{attribute 'GeneratedUsingTerminal: AT2041-0250-0020'}
{attribute addProperty BoxType "AT2041-0250-0020"}
{attribute addProperty Id "A_0102_AT2041_5250_0019_AT2041_5250AT2041_01D6DEDF80"}
{attribute addProperty CRC "3438952946"}
{attribute addProperty Size "80"}
TYPE A_0042_AT2041_0250_0020_CCFA41F2 EXTENDS AT2041_86175B41 :
STRUCT
	{attribute addProperty Name "A_0102_AT2041_5250_0019_AT2041_5250"}
	{attribute addProperty PreviousPort "A_0042(AT2041-0250-0020) : B"}
	A_0102_AT2041_5250_0019_AT2041_5250 : AT2041_01D6DEDF;
END_STRUCT
END_TYPE

(* stored: Version 1.2.0.0, ProductVersion 3.1.4024.9
   DUT A_0042_AT2041_0250_0020_CCFA41F2: Id {79fda706-2ca4-4fc6-8adc-94e8b3447ffd} *)
